// TwinCAT 3 PLC project Cobot_Control
// ProgramVersion: 3.1.4023.0
// libraries:
//   Tc2_EthernetIP, * (Beckhoff Automation GmbH)
//   Tc2_ModbusSrv, * (Beckhoff Automation GmbH)
//   Tc2_Standard, * (Beckhoff Automation GmbH)
//   Tc2_System, * (Beckhoff Automation GmbH)
//   Tc2_Utilities, * (Beckhoff Automation GmbH)
//   Tc3_Module, * (Beckhoff Automation GmbH)
// project tree:
//   GVLs/ E4000_IO.TcGVL, Variables.TcGVL
//   / PlcTask.TcTTO
//   POUs/ Analog_Speed.TcPOU, COMM_FANUC.TcPOU, COMM_UR10.TcPOU, COMPARE_HEXA.TcPOU, Data_Publisher.TcPOU, MAIN.TcPOU, S_Scale.TcPOU
// real-time tasks:
//   TASK PlcTask: cycle T#10ms, priority 20, ADS port 350
//   TASK Task 4: cycle T#1ms, priority 1, ADS port 301
// I/O:
//   DEVICE Device 1 (TC3 EIP Scanner)
//     Box 1 (FANUC Robot R30iB) // <INFO> </INFO> <EDS> C:\TwinCAT\3.1\Config\Io\EtherNetIP\fanucrobot0204_r30ib.eds </EDS>
// variable links:
//   Cobot_Control/Cobot_Control Instance <-> Device 1 (TC3 EIP Scanner)/Box 1 (FANUC Robot R30iB)
//     PlcTask Inputs/Variables.arrFANUC_IN_10[0] <-> Connection 1 (Input/Output)/Inputs/noname0_arrBYTE[31]
//     PlcTask Inputs/Variables.arrFANUC_IN_10[1] <-> Connection 1 (Input/Output)/Inputs/noname0_arrBYTE[32]
//     PlcTask Inputs/Variables.arrFANUC_IN_10[2] <-> Connection 1 (Input/Output)/Inputs/noname0_arrBYTE[33]
//     PlcTask Inputs/Variables.arrFANUC_IN_11[0] <-> Connection 1 (Input/Output)/Inputs/noname0_arrBYTE[34]
//     PlcTask Inputs/Variables.arrFANUC_IN_11[1] <-> Connection 1 (Input/Output)/Inputs/noname0_arrBYTE[35]
//     PlcTask Inputs/Variables.arrFANUC_IN_11[2] <-> Connection 1 (Input/Output)/Inputs/noname0_arrBYTE[36]
//     PlcTask Inputs/Variables.arrFANUC_IN_12[0] <-> Connection 1 (Input/Output)/Inputs/noname0_arrBYTE[37]
//     PlcTask Inputs/Variables.arrFANUC_IN_12[1] <-> Connection 1 (Input/Output)/Inputs/noname0_arrBYTE[38]
//     PlcTask Inputs/Variables.arrFANUC_IN_12[2] <-> Connection 1 (Input/Output)/Inputs/noname0_arrBYTE[39]
//     PlcTask Inputs/Variables.arrFANUC_IN_13[0] <-> Connection 1 (Input/Output)/Inputs/noname0_arrBYTE[40]
//     PlcTask Inputs/Variables.arrFANUC_IN_13[1] <-> Connection 1 (Input/Output)/Inputs/noname0_arrBYTE[41]
//     PlcTask Inputs/Variables.arrFANUC_IN_13[2] <-> Connection 1 (Input/Output)/Inputs/noname0_arrBYTE[42]
//     PlcTask Inputs/Variables.arrFANUC_IN_1[0] <-> Connection 1 (Input/Output)/Inputs/noname0_arrBYTE[3]
//     PlcTask Inputs/Variables.arrFANUC_IN_1[1] <-> Connection 1 (Input/Output)/Inputs/noname0_arrBYTE[4]
//     PlcTask Inputs/Variables.arrFANUC_IN_1[2] <-> Connection 1 (Input/Output)/Inputs/noname0_arrBYTE[5]
//     PlcTask Inputs/Variables.arrFANUC_IN_2[0] <-> Connection 1 (Input/Output)/Inputs/noname0_arrBYTE[6]
//     PlcTask Inputs/Variables.arrFANUC_IN_2[1] <-> Connection 1 (Input/Output)/Inputs/noname0_arrBYTE[7]
//     PlcTask Inputs/Variables.arrFANUC_IN_2[2] <-> Connection 1 (Input/Output)/Inputs/noname0_arrBYTE[8]
//     PlcTask Inputs/Variables.arrFANUC_IN_3[0] <-> Connection 1 (Input/Output)/Inputs/noname0_arrBYTE[9]
//     PlcTask Inputs/Variables.arrFANUC_IN_3[1] <-> Connection 1 (Input/Output)/Inputs/noname0_arrBYTE[10]
//     PlcTask Inputs/Variables.arrFANUC_IN_3[2] <-> Connection 1 (Input/Output)/Inputs/noname0_arrBYTE[11]
//     PlcTask Inputs/Variables.arrFANUC_IN_4[0] <-> Connection 1 (Input/Output)/Inputs/noname0_arrBYTE[12]
//     PlcTask Inputs/Variables.arrFANUC_IN_4[1] <-> Connection 1 (Input/Output)/Inputs/noname0_arrBYTE[13]
//     PlcTask Inputs/Variables.arrFANUC_IN_4[2] <-> Connection 1 (Input/Output)/Inputs/noname0_arrBYTE[14]
//     PlcTask Inputs/Variables.arrFANUC_IN_5[0] <-> Connection 1 (Input/Output)/Inputs/noname0_arrBYTE[15]
//     PlcTask Inputs/Variables.arrFANUC_IN_5[1] <-> Connection 1 (Input/Output)/Inputs/noname0_arrBYTE[16]
//     PlcTask Inputs/Variables.arrFANUC_IN_5[2] <-> Connection 1 (Input/Output)/Inputs/noname0_arrBYTE[17]
//     PlcTask Inputs/Variables.arrFANUC_IN_6[0] <-> Connection 1 (Input/Output)/Inputs/noname0_arrBYTE[18]
//     PlcTask Inputs/Variables.arrFANUC_IN_6[1] <-> Connection 1 (Input/Output)/Inputs/noname0_arrBYTE[19]
//     PlcTask Inputs/Variables.arrFANUC_IN_6[2] <-> Connection 1 (Input/Output)/Inputs/noname0_arrBYTE[20]
//     PlcTask Inputs/Variables.arrFANUC_IN_7[0] <-> Connection 1 (Input/Output)/Inputs/noname0_arrBYTE[22]
//     PlcTask Inputs/Variables.arrFANUC_IN_7[1] <-> Connection 1 (Input/Output)/Inputs/noname0_arrBYTE[23]
//     PlcTask Inputs/Variables.arrFANUC_IN_7[2] <-> Connection 1 (Input/Output)/Inputs/noname0_arrBYTE[24]
//     PlcTask Inputs/Variables.arrFANUC_IN_8[0] <-> Connection 1 (Input/Output)/Inputs/noname0_arrBYTE[25]
//     PlcTask Inputs/Variables.arrFANUC_IN_8[1] <-> Connection 1 (Input/Output)/Inputs/noname0_arrBYTE[26]
//     PlcTask Inputs/Variables.arrFANUC_IN_8[2] <-> Connection 1 (Input/Output)/Inputs/noname0_arrBYTE[27]
//     PlcTask Inputs/Variables.arrFANUC_IN_9[0] <-> Connection 1 (Input/Output)/Inputs/noname0_arrBYTE[28]
//     PlcTask Inputs/Variables.arrFANUC_IN_9[1] <-> Connection 1 (Input/Output)/Inputs/noname0_arrBYTE[29]
//     PlcTask Inputs/Variables.arrFANUC_IN_9[2] <-> Connection 1 (Input/Output)/Inputs/noname0_arrBYTE[30]
//     PlcTask Inputs/Variables.nFANUC_STATE <-> Connection 1 (Input/Output)/Inputs/noname0_arrBYTE[0]
//     PlcTask Outputs/Variables.arrFANUC_OUT_1[0] <-> Connection 1 (Input/Output)/Outputs/noname0_arrBYTE[3]
//     PlcTask Outputs/Variables.arrFANUC_OUT_1[1] <-> Connection 1 (Input/Output)/Outputs/noname0_arrBYTE[4]
//     PlcTask Outputs/Variables.arrFANUC_OUT_1[2] <-> Connection 1 (Input/Output)/Outputs/noname0_arrBYTE[5]

CONFIGURATION Cobot_Control
    RESOURCE PLC ON TwinCAT3
        TASK PlcTask(INTERVAL := T#10ms, PRIORITY := 20);
        PROGRAM MAIN WITH PlcTask : MAIN;
    END_RESOURCE
END_CONFIGURATION

// ---- GVLs/E4000_IO.TcGVL
{attribute 'qualified_only'}
VAR_GLOBAL
	/////////////////////////////////////////////////////////////////////////////////////////////////////////////	
	// Variables for ECCMP88P (1)
	// Digital OUTPUTS
	bSTART_OUT0 AT %Q*: BOOL := FALSE;
	bDIR_IN_OUT1 AT %Q*: BOOL;		
	bUD_IN_OUT2 AT %Q*: BOOL;
	bCNT_IN_OUT3 AT %Q*: BOOL;
	b500_OUT4 AT %Q*: BOOL;		
	bRESET_OUT5 AT %Q*: BOOL;
	bSEL0_OUT6 AT %Q*: BOOL;
	bSEL1_OUT7 AT %Q*: BOOL;		

	// Digital INPUTS
	bRUN_IN0 AT %I*: BOOL;
	bDIR_OUT_IN1 AT %I*: BOOL;
	bCOIN_IN2 AT %I*: BOOL;
	bPULSE_IN3 AT %I*: BOOL;
	bWARNING_IN4 AT %I*: BOOL;
	bERR_IN5 AT %I*: BOOL;

/////////////////////////////////////////////////////////////////////////////////////////////////////////////
	// Variables for ECCMP88P (2)
	// Digital OUTPUTS	
	bEMG_INB_OUT0 AT %Q*: BOOL ;

	// Digital INPUTS
	bMT_CNB_IN0 AT %I*: BOOL;
	bSAFE1B_IN1 AT %I*: BOOL;
	bSAFE2B_IN2 AT %I*: BOOL;
	bAUTO_IN3 AT %I*: BOOL;
	bPWON_IN4 AT %I*: BOOL;

/////////////////////////////////////////////////////////////////////////////////////////////////////////////
	// Variables for ECCEA04 
	// Analog OUTPUT
	nVR AT %Q*: DINT ;
	
	
	// Variables for ECCEA40 
	// Analog INPUTS
	nMOTOR_I_CH0 AT %I*: INT;
	nLOAD_CH1 AT %I*: INT;
	nSPEED_V_CH2 AT %I*: INT;
	
/////////////////////////////////////////////////////////////////////////////////////////////////////////////
	// Variables to help control
	
	bSetSpeed : BOOL := FALSE;
	
	
	
	

END_VAR

// ---- GVLs/Variables.TcGVL
{attribute 'qualified_only'}
VAR_GLOBAL
	
	////////////////////////////////////////////////////////////////////////
	// Variables for ModBUS TCP to connect, monitor and control UR robots //
	mb_Input_Coils AT %I* : ARRAY [0..255] OF BOOL;
	mb_Output_Coils : ARRAY [0..255] OF BOOL;
	mb_Input_Registers : ARRAY [0..255] OF WORD;
	mb_Output_Registers : ARRAY [0..255] OF WORD;	
	////////////////////////////////////////////////////////////////////////

	{attribute 'OPC.UA.DA.Access' := '3'}
	{attribute 'OPC.UA.DA' := '1'}
	bStartStop AT %I* : BOOL;	

	////////////////////////////// UR Robot ///////////////////////////////
	
	///////////////////	 Raw UR Robot Information  ////////////////////////
	
	arrURAngles AT %I*          	: ARRAY [1..6] OF INT;
	arrURAnglesVelocity AT %I*     	: ARRAY [1..6] OF INT;	
	arrURAnglesCurrent AT %I*      	: ARRAY [1..6] OF INT;		
	arrURAnglesTemp AT %I*        	: ARRAY [1..6] OF INT;		
	arrURJointMode AT %I*        	: ARRAY [1..6] OF INT;	
	arrTCPCartData AT %I*          	: ARRAY [1..3] OF INT;	
	arrTCPRotData AT %I*          	: ARRAY [1..3] OF INT;	
	arrURRobotStatus AT%I*			: ARRAY [1..6] OF INT;
	nURProgState 					: INT;
	nURProgAction  					: INT;		
	nPLCProgState  					: INT;
		
	/////////////////////////////////////////////////////////////////////////	

	///////////////////	 Transformed UR Robot Information  ///////////////////
	{attribute 'OPC.UA.DA' := '1'}
	arrfUR_TCPxyz AT %Q* 			: ARRAY[1..3] OF REAL ;	
	{attribute 'OPC.UA.DA' := '1'}
	arrfUR_TCPuvw AT %Q* 			: ARRAY[1..3] OF REAL ;
	{attribute 'OPC.UA.DA' := '1'}
	arrfUR_Angles AT %Q* 			: ARRAY[1..6] OF REAL ;
	{attribute 'OPC.UA.DA' := '1'}
	arrfUR_AnglesVel AT %Q* 		: ARRAY[1..6] OF REAL ;
	{attribute 'OPC.UA.DA' := '1'}
	arrfUR_AnglesAmp AT %Q* 		: ARRAY[1..6] OF REAL ;
	{attribute 'OPC.UA.DA' := '1'}
	arrfUR_AnglesTemp AT %Q* 		: ARRAY[1..6] OF REAL ;
	{attribute 'OPC.UA.DA' := '1'}
	arrfUR_JntMode AT %Q* 			: ARRAY[1..6] OF REAL ;
	{attribute 'OPC.UA.DA' := '1'}
	arrfUR_Status AT %Q* 			: ARRAY[1..6] OF REAL ;

	///////////////////////////////////////////////////////////////////////////
	
	
	
	////////////////////////////// FANUC Robot /////////////////////////////
	
	///////////////////	 Raw FANUC Robot Information  ///////////////////

	nFANUC_STATE  AT %I*         	: UINT;
	
	arrFANUC_IN_1 AT %I*	       	: ARRAY [0..2] OF UINT; // Starts at 3
	arrFANUC_IN_2 AT %I* 		  	: ARRAY [0..2] OF UINT;	
	arrFANUC_IN_3 AT %I*  	    	: ARRAY [0..2] OF UINT;		
	arrFANUC_IN_4 AT %I* 			: ARRAY [0..2] OF UINT;	
	arrFANUC_IN_5 AT %I*  		  	: ARRAY [0..2] OF UINT;		
	arrFANUC_IN_6 AT %I* 			: ARRAY [0..2] OF UINT;	
	arrFANUC_IN_7 AT %I*	       	: ARRAY [0..2] OF UINT; // Starts at 22
	arrFANUC_IN_8 AT %I* 		  	: ARRAY [0..2] OF UINT;	
	arrFANUC_IN_9 AT %I*  	    	: ARRAY [0..2] OF UINT;		
	arrFANUC_IN_10 AT %I* 			: ARRAY [0..2] OF UINT;	
	arrFANUC_IN_11 AT %I*  		  	: ARRAY [0..2] OF UINT;		
	arrFANUC_IN_12 AT %I* 			: ARRAY [0..2] OF UINT;	
	arrFANUC_IN_13 AT %I* 			: ARRAY [0..2] OF UINT;
	
	nFANUC_REMOTE_START	AT %Q*		: UINT := 0;
	
	arrFANUC_OUT_1 AT %Q*  			: ARRAY [0..2] OF UINT;	
	arrFANUC_OUT_2          		: ARRAY [0..2] OF UINT;	
	arrFANUC_OUT_3           		: ARRAY [0..2] OF UINT;	
	arrFANUC_OUT_4 					: ARRAY [0..2] OF UINT;	
	arrFANUC_OUT_5          	 	: ARRAY [0..2] OF UINT;	
	arrFANUC_OUT_6 					: ARRAY [0..2] OF UINT;		
	arrFANUC_OUT_7        			: ARRAY [0..2] OF UINT;	
	arrFANUC_OUT_8          		: ARRAY [0..2] OF UINT;	
	arrFANUC_OUT_9           		: ARRAY [0..2] OF UINT;	
	arrFANUC_OUT_10					: ARRAY [0..2] OF UINT;	
	arrFANUC_OUT_11          	 	: ARRAY [0..2] OF UINT;	
	arrFANUC_OUT_12					: ARRAY [0..2] OF UINT;	
	
	///////////////////////////////////////////////////////////
	
	///////////////////	 Transformed FANUC Robot Information  ///////////////////
	{attribute 'OPC.UA.DA' := '1'}
	arrfFANUC_TCPxyz AT %Q* 		: ARRAY[1..3] OF REAL ;	
	{attribute 'OPC.UA.DA' := '1'}
	arrfFANUC_TCPuvw AT %Q* 		: ARRAY[1..3] OF REAL ;
	{attribute 'OPC.UA.DA' := '1'}
	arrfFANUC_Angles AT %Q* 		: ARRAY[1..6] OF REAL ;

	///////////////////////////////////////////////////////////////////////////
	
END_VAR

// ---- POUs/MAIN.TcPOU
PROGRAM MAIN
VAR		
	bStartProcess 	: BOOL := FALSE;
	timer1			: TON;
	timer2			: TON;
	timer3			: TON;
	bStart1			: BOOL := FALSE;
	bStart2: BOOL;
	bStart3: BOOL;
END_VAR

// Beginning of painting process //

// If process is initiated from UI
IF (bStartProcess) THEN
	bStart1 := TRUE;
	timer1(IN := bStart1, PT:= T#5S);
		
	IF timer1.Q THEN		
		Variables.nFANUC_REMOTE_START := 160; // Initializing variables #6 (Starts)
		bStart2 := TRUE;
	END_IF
	
	COMM_FANUC.arrf_Internal_FANUC_Output_1 := 63; // Tell FANUC to move and leave robot in initial position	
	
	timer2(IN := bStart2, PT:= T#1S);
		
	IF timer2.Q THEN		
		Variables.nFANUC_REMOTE_START := 128; // Start works in a rising edge
	END_IF
	
	
	IF COMM_FANUC.arrf_Internal_FANUC_Input_1 = 254 THEN // IF FANUC tells us that position has been reached, we proceed to move UR
		Variables.nURProgAction := 63; // Set Program in UR - Move Robot		
		// Wait for UR to finish
		
		IF Variables.nURProgState = 99 THEN // If UR finishes
			COMM_FANUC.arrf_Internal_FANUC_Output_1 := 77; // Inform FANUC that it is safe to move home
			bStart3 := TRUE;			
			timer3(IN := bStart3, PT:= T#3S);			
			IF timer3.Q THEN
				
				bStartProcess := FALSE; // Terminate process
			END_IF
								
		END_IF		
	END_IF

ELSE // IF not initiated
	// While no signal for starting demo is coming, set variables of robots as 0
	//timer1.IN := FALSE;
	//Variables.nFANUC_REMOTE_START := 0;
	COMM_FANUC.arrf_Internal_FANUC_Output_1 := 0;
	Variables.nURProgAction := 0;
	Variables.nFANUC_REMOTE_START := 128; // Initializing variables #8 (Enable function)
	bStart1 := FALSE;
	bStart2 := FALSE;
	bStart3 := FALSE;
	timer1(IN:=bStart1);
	timer2(IN:=bStart2);
	timer3(IN:=bStart3);
END_IF


Data_Publisher();
COMM_UR10();
COMM_FANUC();
Analog_Speed();

END_PROGRAM

// ---- POUs/COMM_FANUC.TcPOU
{attribute 'qualified_only}
PROGRAM COMM_FANUC

VAR_INPUT    
	arrf_Internal_FANUC_Input_1			: REAL;
	arrf_Internal_FANUC_Output_1		: UINT;
	
END_VAR

VAR_OUTPUT	
	
	sOutput_String						: STRING;
END_VAR

VAR		
	arrf_Internal_FANUC_TCP_xyz			: ARRAY [1..3] OF REAL;
	arrf_Internal_FANUC_TCP_uvw			: ARRAY [1..3] OF REAL;
	arrf_Internal_FANUC_TCP_Joints		: ARRAY [1..6] OF REAL;	
	fbCOMPARE_HEXA: COMPARE_HEXA;
END_VAR

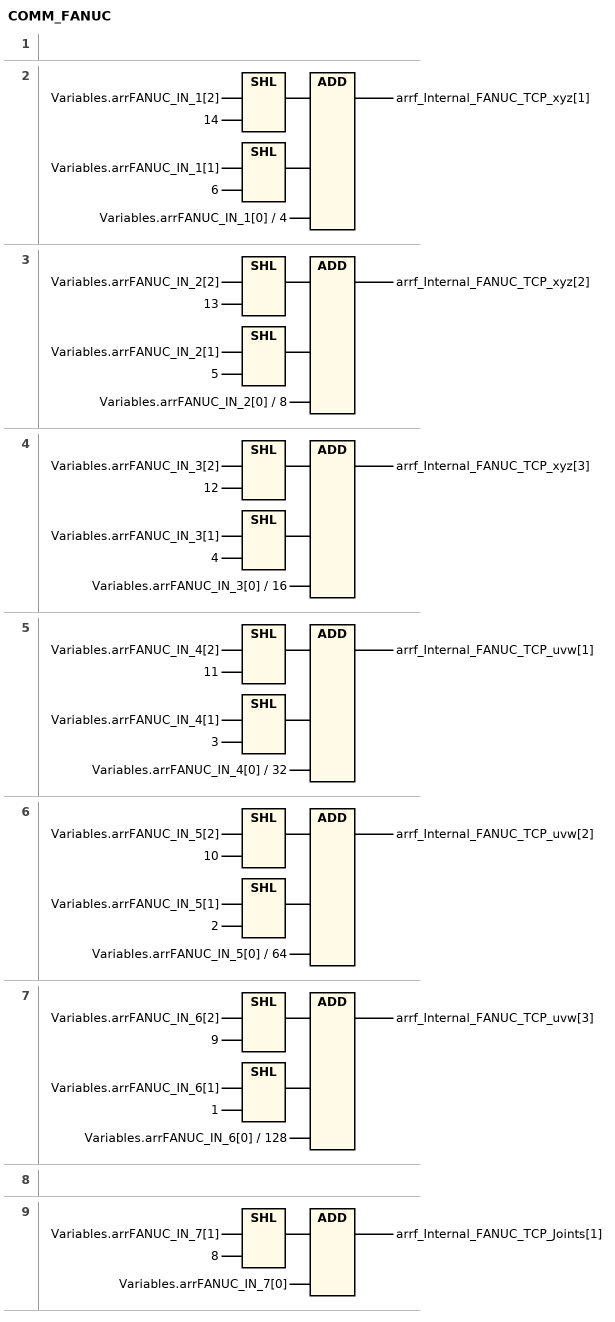
// NETWORK 1

// NETWORK 2
arrf_Internal_FANUC_TCP_xyz[1] := SHL(Variables.arrFANUC_IN_1[2], 14) + SHL(Variables.arrFANUC_IN_1[1], 6) + (Variables.arrFANUC_IN_1[0] / 4);

// NETWORK 3
arrf_Internal_FANUC_TCP_xyz[2] := SHL(Variables.arrFANUC_IN_2[2], 13) + SHL(Variables.arrFANUC_IN_2[1], 5) + (Variables.arrFANUC_IN_2[0] / 8);

// NETWORK 4
arrf_Internal_FANUC_TCP_xyz[3] := SHL(Variables.arrFANUC_IN_3[2], 12) + SHL(Variables.arrFANUC_IN_3[1], 4) + (Variables.arrFANUC_IN_3[0] / 16);

// NETWORK 5
arrf_Internal_FANUC_TCP_uvw[1] := SHL(Variables.arrFANUC_IN_4[2], 11) + SHL(Variables.arrFANUC_IN_4[1], 3) + (Variables.arrFANUC_IN_4[0] / 32);

// NETWORK 6
arrf_Internal_FANUC_TCP_uvw[2] := SHL(Variables.arrFANUC_IN_5[2], 10) + SHL(Variables.arrFANUC_IN_5[1], 2) + (Variables.arrFANUC_IN_5[0] / 64);

// NETWORK 7
arrf_Internal_FANUC_TCP_uvw[3] := SHL(Variables.arrFANUC_IN_6[2], 9) + SHL(Variables.arrFANUC_IN_6[1], 1) + (Variables.arrFANUC_IN_6[0] / 128);

// NETWORK 8

// NETWORK 9
arrf_Internal_FANUC_TCP_Joints[1] := SHL(Variables.arrFANUC_IN_7[1], 8) + Variables.arrFANUC_IN_7[0];

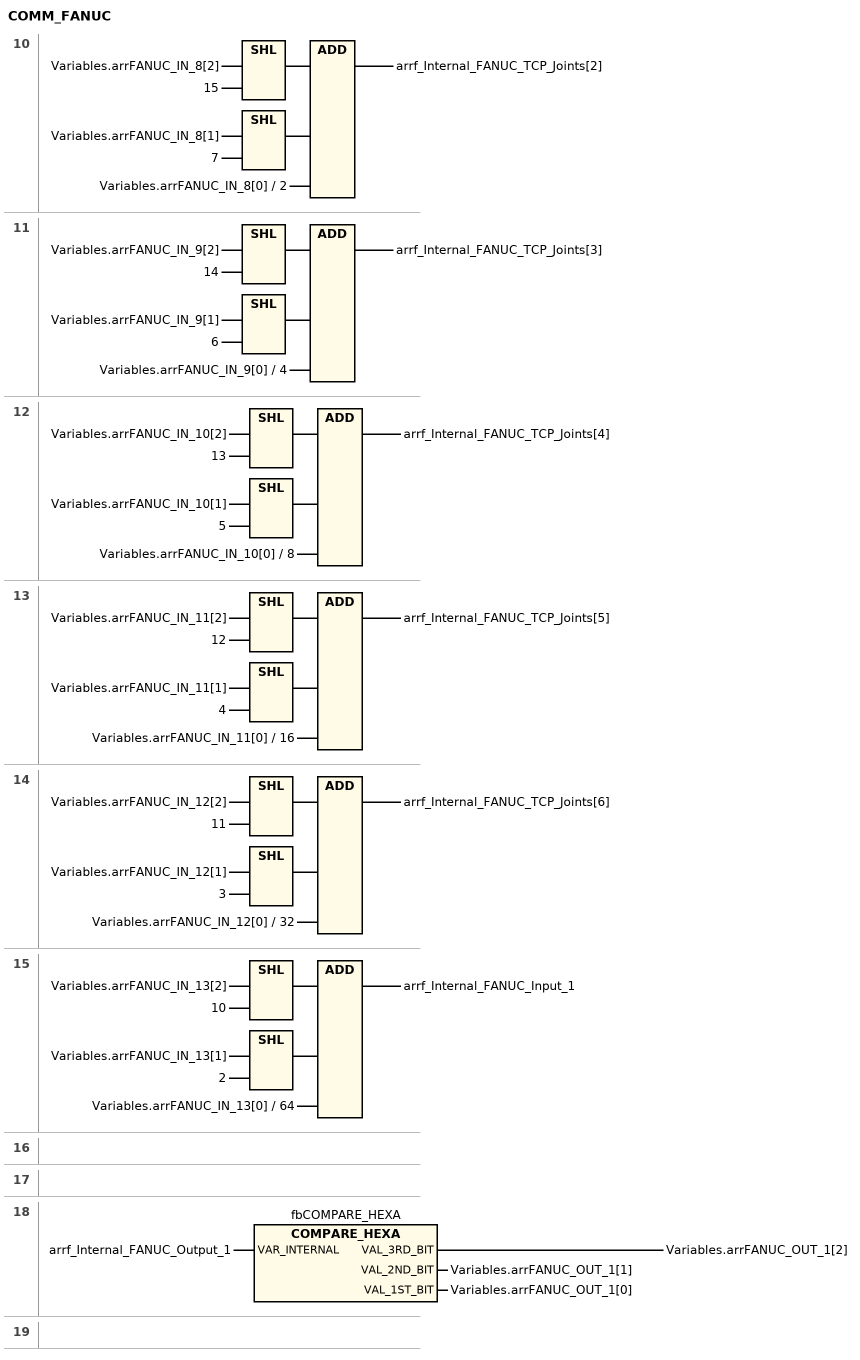
// NETWORK 10
arrf_Internal_FANUC_TCP_Joints[2] := SHL(Variables.arrFANUC_IN_8[2], 15) + SHL(Variables.arrFANUC_IN_8[1], 7) + (Variables.arrFANUC_IN_8[0] / 2);

// NETWORK 11
arrf_Internal_FANUC_TCP_Joints[3] := SHL(Variables.arrFANUC_IN_9[2], 14) + SHL(Variables.arrFANUC_IN_9[1], 6) + (Variables.arrFANUC_IN_9[0] / 4);

// NETWORK 12
arrf_Internal_FANUC_TCP_Joints[4] := SHL(Variables.arrFANUC_IN_10[2], 13) + SHL(Variables.arrFANUC_IN_10[1], 5) + (Variables.arrFANUC_IN_10[0] / 8);

// NETWORK 13
arrf_Internal_FANUC_TCP_Joints[5] := SHL(Variables.arrFANUC_IN_11[2], 12) + SHL(Variables.arrFANUC_IN_11[1], 4) + (Variables.arrFANUC_IN_11[0] / 16);

// NETWORK 14
arrf_Internal_FANUC_TCP_Joints[6] := SHL(Variables.arrFANUC_IN_12[2], 11) + SHL(Variables.arrFANUC_IN_12[1], 3) + (Variables.arrFANUC_IN_12[0] / 32);

// NETWORK 15
arrf_Internal_FANUC_Input_1 := SHL(Variables.arrFANUC_IN_13[2], 10) + SHL(Variables.arrFANUC_IN_13[1], 2) + (Variables.arrFANUC_IN_13[0] / 64);

// NETWORK 16

// NETWORK 17

// NETWORK 18
fbCOMPARE_HEXA(
    VAR_INTERNAL := arrf_Internal_FANUC_Output_1,
    VAL_2ND_BIT => Variables.arrFANUC_OUT_1[1],
    VAL_1ST_BIT => Variables.arrFANUC_OUT_1[0]); // COMPARE_HEXA
Variables.arrFANUC_OUT_1[2] := fbCOMPARE_HEXA.VAL_3RD_BIT;

// NETWORK 19

END_PROGRAM

// ---- POUs/COMPARE_HEXA.TcPOU
FUNCTION_BLOCK COMPARE_HEXA
VAR_INPUT
	VAR_INTERNAL : UINT;
END_VAR
VAR_OUTPUT
	Error		 : BOOL;
	VAL_3RD_BIT	 : UINT;
	VAL_2ND_BIT	 : UINT;
	VAL_1ST_BIT	 : UINT;
END_VAR
VAR	
END_VAR

IF VAR_INTERNAL >= 16384 AND VAR_INTERNAL < 65356 THEN	
	VAL_3RD_BIT := VAR_INTERNAL/16384;	
	VAL_2ND_BIT := (VAR_INTERNAL - (16384*VAL_3RD_BIT))/64;
	VAL_1ST_BIT := (VAR_INTERNAL - (16384*VAL_3RD_BIT) - (64*VAL_2ND_BIT))*4;
END_IF	
IF VAR_INTERNAL >= 64 AND VAR_INTERNAL < 16384 THEN
	VAL_3RD_BIT := 0;	
	VAL_2ND_BIT := VAR_INTERNAL/64;
	VAL_1ST_BIT := (VAR_INTERNAL - (64*VAL_2ND_BIT))*4;		
END_IF
IF VAR_INTERNAL >= 0 AND VAR_INTERNAL < 64 THEN
	VAL_3RD_BIT := 0;		
	VAL_2ND_BIT := 0;
	VAL_1ST_BIT := VAR_INTERNAL*4;		
END_IF

END_FUNCTION_BLOCK

// ---- POUs/Data_Publisher.TcPOU
PROGRAM Data_Publisher
VAR
	i : INT := 1;
	j : INT := 1;
	k : INT := 1;
END_VAR

i := 1;
j := 1;

///////////////////////////////////////////////////////////////////////////////////////////

// UR updates //

IF NOT COMM_UR10.bError1  THEN	
	FOR i := 1 TO 3 BY 1 DO
		Variables.arrfUR_TCPxyz[i] := INT_TO_REAL(Variables.arrTCPCartData[i])/(10);	
		Variables.arrfUR_TCPuvw[i] := INT_TO_REAL(Variables.arrTCPRotData[i])/(1000);
	END_FOR	
	i := 1;
ELSE
	FOR i := 1 TO 3 BY 1 DO
		Variables.arrfUR_TCPxyz[i] := 0;	
		Variables.arrfUR_TCPuvw[i] := 0;
	END_FOR	
	i := 1;	
END_IF

IF NOT COMM_UR10.bError2  THEN
	FOR j := 1 TO 6 BY 1 DO
		Variables.arrfUR_Angles[j] := INT_TO_REAL(Variables.arrURAngles[j])/(17.444);	
		Variables.arrfUR_AnglesVel[j] := INT_TO_REAL(Variables.arrURAnglesVelocity[j]);
		Variables.arrfUR_AnglesAmp[j] := INT_TO_REAL(Variables.arrURAnglesCurrent[j]);	
		Variables.arrfUR_AnglesTemp[j] := INT_TO_REAL(Variables.arrURAnglesTemp[j]);
		Variables.arrfUR_JntMode[j] := INT_TO_REAL(Variables.arrURJointMode[j]);	
		Variables.arrfUR_Status[j] := INT_TO_REAL(Variables.arrURRobotStatus[j]);
	END_FOR
	j := 1;
ELSE
	FOR j := 1 TO 6 BY 1 DO
		Variables.arrfUR_Angles[j] := 0;	
		Variables.arrfUR_AnglesVel[j] := 0;
		Variables.arrfUR_AnglesAmp[j] := 0;	
		Variables.arrfUR_AnglesTemp[j] := 0;
		Variables.arrfUR_JntMode[j] := 0;	
		Variables.arrfUR_Status[j] := 0;
	END_FOR
	j := 1;
END_IF

///////////////////////////////////////////////////////////////////////////////////////////

// Fanuc Updates //
k := 1;
FOR k := 1 TO 3 BY 1 DO
	IF COMM_FANUC.arrf_Internal_FANUC_TCP_xyz[k] > 32676 THEN
		Variables.arrfFANUC_TCPxyz[k] := ((65535 - COMM_FANUC.arrf_Internal_FANUC_TCP_xyz[k]) / 10);
	ELSE
		Variables.arrfFANUC_TCPxyz[k] := COMM_FANUC.arrf_Internal_FANUC_TCP_xyz[k] / 10;		
	END_IF
END_FOR

k := 1;
FOR k := 1 TO 3 BY 1 DO
	IF COMM_FANUC.arrf_Internal_FANUC_TCP_uvw[k] > 32676 THEN
		Variables.arrfFANUC_TCPuvw[k] := ((65535 - COMM_FANUC.arrf_Internal_FANUC_TCP_uvw[k]) / 10);
	ELSE
		Variables.arrfFANUC_TCPuvw[k] := COMM_FANUC.arrf_Internal_FANUC_TCP_uvw[k] / 10;		
	END_IF
END_FOR

k := 1;
FOR k := 1 TO 6 BY 1 DO
	IF COMM_FANUC.arrf_Internal_FANUC_TCP_Joints[k] > 32676 THEN
		Variables.arrfFANUC_Angles[k] := ((65535 - COMM_FANUC.arrf_Internal_FANUC_TCP_Joints[k]) / 100);
	ELSE
		Variables.arrfFANUC_Angles[k] := COMM_FANUC.arrf_Internal_FANUC_TCP_Joints[k] / 100;		
	END_IF
END_FOR


///////////////////////////////////////////////////////////////////////////////////////////

END_PROGRAM

// ---- POUs/COMM_UR10.TcPOU
{attribute 'qualified_only}
PROGRAM COMM_UR10
VAR
	FB1: FB_MBReadRegs;
	
	// IP address & Port of ModBUS Server //
	ipAddr         					: STRING(15) := '192.168.1.13';
	iMBPort							: UINT := 502;
	
	// Function Blocks to extract robot information //
	// UR Robot Addresses and Array Sizes //
	nAddrrToolTCPCart				: WORD := 400;
	nAddrrToolTCPRot				: WORD := 403;
	nAddrrURAngles					: WORD := 270;
	nAddrrURAnglesVelocity			: WORD := 280;
	nAddrrURAnglesCurrent			: WORD := 290;
	nAddrrURAnglesTemp				: WORD := 300;
	nAddrrURJointMode				: WORD := 310;	
	nAddrrURState					: WORD := 260;
	nAddrrURProgAction				: WORD := 136;
	nAddrrURProgState				: WORD := 128;
	nAddrrPLCProgState				: WORD := 137;
	
	nQtyUnit						: WORD := 1;
	nQtyCart						: WORD := 3;
	nQtyRot							: WORD := 3;	
	nQtyURAxes						: WORD := 6;
		
	
	// Blocks //
	
	// Robot Angles information //	
	fbURAngles						: FB_MBReadRegs;
	// Robot Angles Velocity information //	
	fbURAnglesVelocity				: FB_MBReadRegs;
	// Robot Angles Current information //	
	fbURAnglesCurrent				: FB_MBReadRegs;
	// Robot Angles Temperature information //	
	fbURAnglesTemp					: FB_MBReadRegs;
	// Robot Joint Mode information //	
	fbURJointMode					: FB_MBReadRegs;
	// Robot Tool TCP Cart //	
	fbTool_TCP_Cartesian			: FB_MBReadRegs;
	// Robot Tool TCP Rot //
	fbTool_TCP_Rotation				: FB_MBReadRegs;
	// Robot Status //
	fbURRobot_Status				: FB_MBReadRegs;
	
	// Robot program start //
	fbURprogram_start				: FB_MBWriteRegs;
	// Robot state in program //
	fbUR_state_in_program			: FB_MBReadRegs;
	// PLC state in program //
	fbPLC_state_in_program			: FB_MBWriteRegs;
	
		
	// Reading Register - FB //
	fbReadRegs						: FB_MBReadRegs;
	bReadRegs						: BOOL;
	bReadRegsBusy   				: BOOL;
	bReadRegsError  				: BOOL;
	nReadRegsErrorId        		: UDINT;	
	
	// Writing Register - FB //
	fbWriteRegs						: FB_MBWriteRegs;
	bWriteRegs						: BOOL;
	bWriteRegsBusy   				: BOOL;
	bWriteRegsError  				: BOOL;
	nWriteRegsErrorId        		: UDINT;	
	
	// Error Variables //
	bError1, bError2, bError3		: BOOL;
	nErrID1, nErrID2, nErrID3		: UDINT;
	cbRead1, cbRead2, cbRead3		: UDINT;
	
	// Timers //
	TONreaders						: TON;
	TONwriters						: TON;
	tRefresh						: TIME := T#0.5S;
	tGiveUp							: TIME := T#2S;	
	
END_VAR

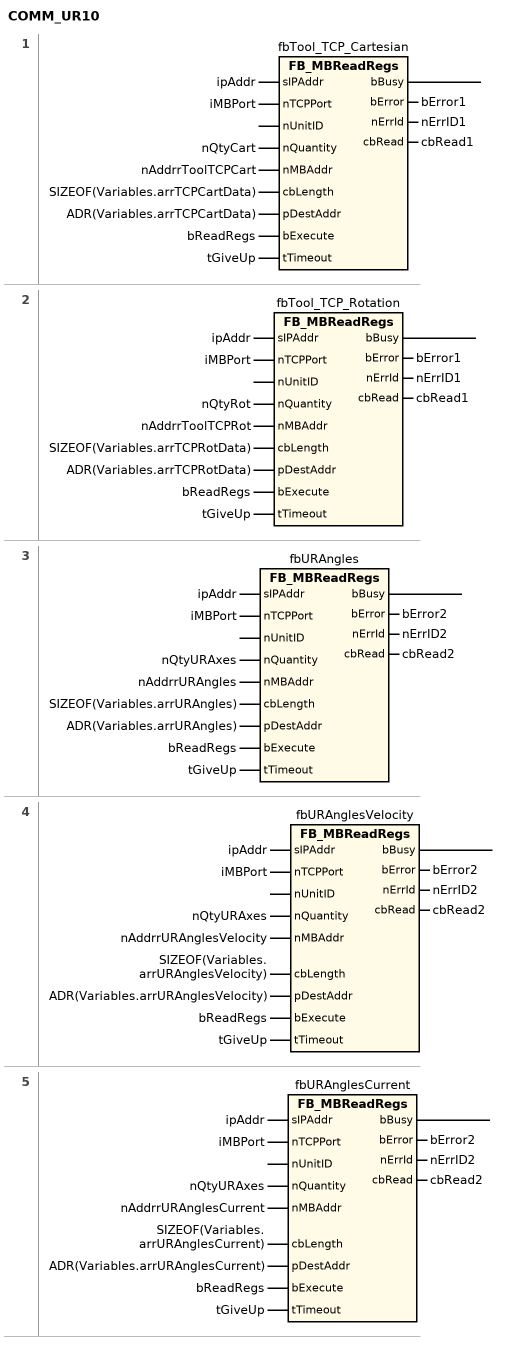
// NETWORK 1
fbTool_TCP_Cartesian(
    sIPAddr := ipAddr,
    nTCPPort := iMBPort,
    nQuantity := nQtyCart,
    nMBAddr := nAddrrToolTCPCart,
    cbLength := SIZEOF(Variables.arrTCPCartData),
    pDestAddr := ADR(Variables.arrTCPCartData),
    bExecute := bReadRegs,
    tTimeout := tGiveUp,
    bError => bError1,
    nErrId => nErrID1,
    cbRead => cbRead1); // FB_MBReadRegs

// NETWORK 2
fbTool_TCP_Rotation(
    sIPAddr := ipAddr,
    nTCPPort := iMBPort,
    nQuantity := nQtyRot,
    nMBAddr := nAddrrToolTCPRot,
    cbLength := SIZEOF(Variables.arrTCPRotData),
    pDestAddr := ADR(Variables.arrTCPRotData),
    bExecute := bReadRegs,
    tTimeout := tGiveUp,
    bError => bError1,
    nErrId => nErrID1,
    cbRead => cbRead1); // FB_MBReadRegs

// NETWORK 3
fbURAngles(
    sIPAddr := ipAddr,
    nTCPPort := iMBPort,
    nQuantity := nQtyURAxes,
    nMBAddr := nAddrrURAngles,
    cbLength := SIZEOF(Variables.arrURAngles),
    pDestAddr := ADR(Variables.arrURAngles),
    bExecute := bReadRegs,
    tTimeout := tGiveUp,
    bError => bError2,
    nErrId => nErrID2,
    cbRead => cbRead2); // FB_MBReadRegs

// NETWORK 4
fbURAnglesVelocity(
    sIPAddr := ipAddr,
    nTCPPort := iMBPort,
    nQuantity := nQtyURAxes,
    nMBAddr := nAddrrURAnglesVelocity,
    cbLength := SIZEOF(Variables.arrURAnglesVelocity),
    pDestAddr := ADR(Variables.arrURAnglesVelocity),
    bExecute := bReadRegs,
    tTimeout := tGiveUp,
    bError => bError2,
    nErrId => nErrID2,
    cbRead => cbRead2); // FB_MBReadRegs

// NETWORK 5
fbURAnglesCurrent(
    sIPAddr := ipAddr,
    nTCPPort := iMBPort,
    nQuantity := nQtyURAxes,
    nMBAddr := nAddrrURAnglesCurrent,
    cbLength := SIZEOF(Variables.arrURAnglesCurrent),
    pDestAddr := ADR(Variables.arrURAnglesCurrent),
    bExecute := bReadRegs,
    tTimeout := tGiveUp,
    bError => bError2,
    nErrId => nErrID2,
    cbRead => cbRead2); // FB_MBReadRegs

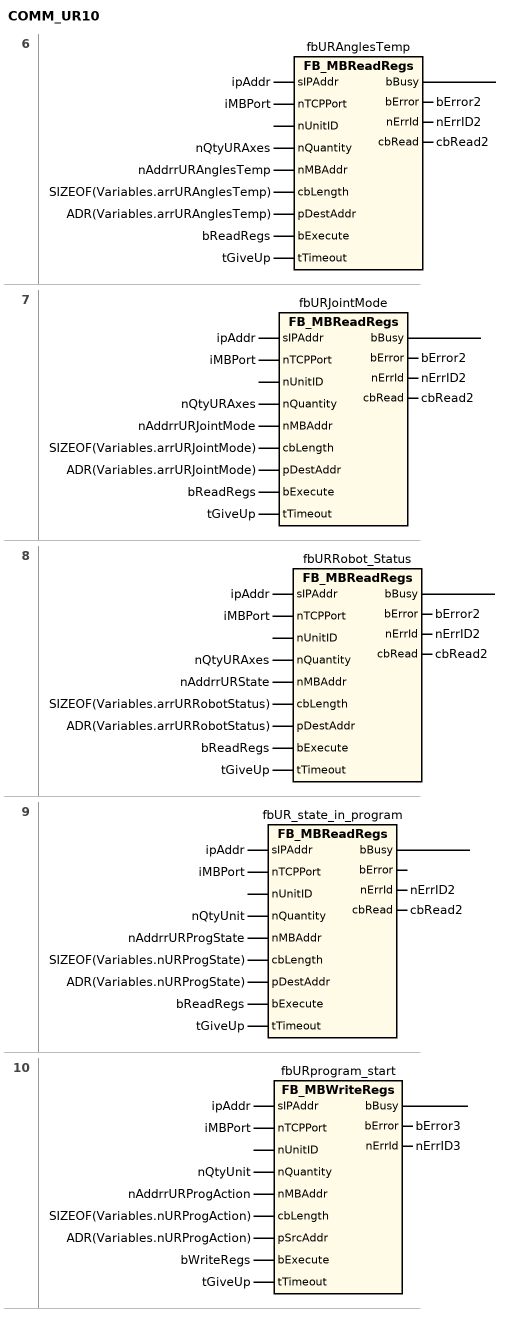
// NETWORK 6
fbURAnglesTemp(
    sIPAddr := ipAddr,
    nTCPPort := iMBPort,
    nQuantity := nQtyURAxes,
    nMBAddr := nAddrrURAnglesTemp,
    cbLength := SIZEOF(Variables.arrURAnglesTemp),
    pDestAddr := ADR(Variables.arrURAnglesTemp),
    bExecute := bReadRegs,
    tTimeout := tGiveUp,
    bError => bError2,
    nErrId => nErrID2,
    cbRead => cbRead2); // FB_MBReadRegs

// NETWORK 7
fbURJointMode(
    sIPAddr := ipAddr,
    nTCPPort := iMBPort,
    nQuantity := nQtyURAxes,
    nMBAddr := nAddrrURJointMode,
    cbLength := SIZEOF(Variables.arrURJointMode),
    pDestAddr := ADR(Variables.arrURJointMode),
    bExecute := bReadRegs,
    tTimeout := tGiveUp,
    bError => bError2,
    nErrId => nErrID2,
    cbRead => cbRead2); // FB_MBReadRegs

// NETWORK 8
fbURRobot_Status(
    sIPAddr := ipAddr,
    nTCPPort := iMBPort,
    nQuantity := nQtyURAxes,
    nMBAddr := nAddrrURState,
    cbLength := SIZEOF(Variables.arrURRobotStatus),
    pDestAddr := ADR(Variables.arrURRobotStatus),
    bExecute := bReadRegs,
    tTimeout := tGiveUp,
    bError => bError2,
    nErrId => nErrID2,
    cbRead => cbRead2); // FB_MBReadRegs

// NETWORK 9
fbUR_state_in_program(
    sIPAddr := ipAddr,
    nTCPPort := iMBPort,
    nQuantity := nQtyUnit,
    nMBAddr := nAddrrURProgState,
    cbLength := SIZEOF(Variables.nURProgState),
    pDestAddr := ADR(Variables.nURProgState),
    bExecute := bReadRegs,
    tTimeout := tGiveUp,
    nErrId => nErrID2,
    cbRead => cbRead2); // FB_MBReadRegs

// NETWORK 10
fbURprogram_start(
    sIPAddr := ipAddr,
    nTCPPort := iMBPort,
    nQuantity := nQtyUnit,
    nMBAddr := nAddrrURProgAction,
    cbLength := SIZEOF(Variables.nURProgAction),
    pSrcAddr := ADR(Variables.nURProgAction),
    bExecute := bWriteRegs,
    tTimeout := tGiveUp,
    bError => bError3,
    nErrId => nErrID3); // FB_MBWriteRegs

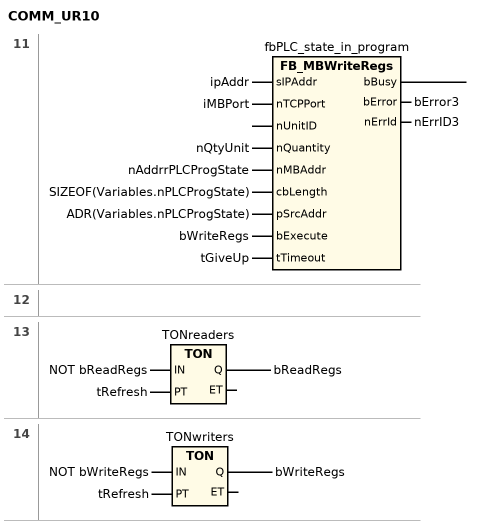
// NETWORK 11
fbPLC_state_in_program(
    sIPAddr := ipAddr,
    nTCPPort := iMBPort,
    nQuantity := nQtyUnit,
    nMBAddr := nAddrrPLCProgState,
    cbLength := SIZEOF(Variables.nPLCProgState),
    pSrcAddr := ADR(Variables.nPLCProgState),
    bExecute := bWriteRegs,
    tTimeout := tGiveUp,
    bError => bError3,
    nErrId => nErrID3); // FB_MBWriteRegs

// NETWORK 12

// NETWORK 13
TONreaders(IN := NOT bReadRegs, PT := tRefresh); // TON
bReadRegs := TONreaders.Q;

// NETWORK 14
TONwriters(IN := NOT bWriteRegs, PT := tRefresh); // TON
bWriteRegs := TONwriters.Q;

END_PROGRAM

// ---- POUs/Analog_Speed.TcPOU
PROGRAM Analog_Speed
VAR
	fScaledSpeed				:DINT;
END_VAR

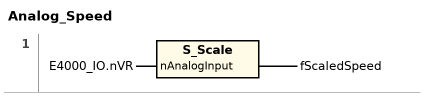
// NETWORK 1
fScaledSpeed := S_Scale(nAnalogInput := E4000_IO.nVR);

END_PROGRAM

// ---- POUs/S_Scale.TcPOU
FUNCTION S_Scale : DINT
VAR_INPUT
	nAnalogInput : DINT;
END_VAR
VAR
END_VAR

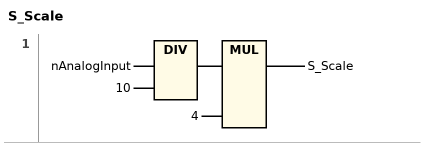
// NETWORK 1
S_Scale := (nAnalogInput / 10) * 4;

END_FUNCTION
